// TwinCAT 3 PLC project TcoDrivesBeckhoff
// Title: TcoDrivesBeckhoff
// Company: Vortex.Library
// Author: TcOpenGroup
// ProjectVersion: 0.6.0.913
// ProgramVersion: 3.1.4024.12
// libraries:
//   Tc2_MC2, * (Beckhoff Automation GmbH)
//   Tc2_MC2_Drive, * (Beckhoff Automation GmbH)
//   Tc2_NCI, * (Beckhoff Automation GmbH)
//   Tc2_Standard, * (Beckhoff Automation GmbH)
//   Tc2_System, * (Beckhoff Automation GmbH)
//   Tc2_Utilities, * (Beckhoff Automation GmbH)
//   Tc3_Module, * (Beckhoff Automation GmbH)
//   TcoCore, 0.6.0.913 (Vortex.Library)
// project tree:
//   DUTs/ eAxisParameter.TcDUT (not stored), eAxisEncoderReferenceSystem.TcDUT (not stored), eDirection.TcDUT (not stored), eAxisStates.TcDUT (not stored), eEncoderReferenceMode.TcDUT (not stored), eHomingMode.TcDUT (not stored), ePowerOverride.TcDUT (not stored), eSetPositionMode.TcDUT (not stored), eJogMode.TcDUT (not stored), TcoAxisOpModes.TcDUT (not stored), TcoAxisRef.TcPOU (not stored), TcoAxisStatus.TcDUT (not stored), TcoAxisConfig.TcDUT (not stored)
//   DUTs/Interpolator/HW/ TcoGenericInterpolatorHw.TcDUT, TcoGenericInterpolatorHwInputs.TcDUT, TcoGenericInterpolatorHwOutputs.TcDUT
//   DUTs/Interpolator/ TcoGenericInterpolatorData.TcDUT
//   / PlcTask.TcTTO (not stored)
//   POUs/Conversions/ Tc2MC2_TO_Tco_AxisStates.TcPOU (not stored), LREAL_TO_Tco_AxisEncoderReferenceSystem.TcPOU (not stored), Tc2MC2_TO_Tco_SetPositionMode.TcPOU (not stored), Tc2MC2_TO_Tco_JogMode.TcPOU (not stored), Tco_TO_Tc2MC2_SetPositionMode.TcPOU (not stored), Tco_TO_Tc2MC2_Direction.TcPOU (not stored), Tc2MC2_TO_Tco_Direction.TcPOU (not stored), Tco_TO_Tc2MC2_HomingMode.TcPOU (not stored), Tco_TO_Tc2MC2_EncRefMode.TcPOU (not stored), Tc2MC2_TO_Tco_EncRefMode.TcPOU (not stored), Tc2MC2_TO_Tco_HomingMode.TcPOU (not stored), Tco_TO_Tc2MC2_AxisStates.TcPOU (not stored), Tco_TO_Tc2MC2_JogMode.TcPOU (not stored)
//   POUs/ MAIN.TcPOU (not stored)
//   POUs/Prototypes/CartesianCoordinateSystem/Intetrpolator/ TcoInterpolator.TcPOU, TcoInterpolatorConfig.TcDUT, TcoInterpolatorStatus.TcDUT, TcoInterpolatorControl.TcDUT
//   POUs/Prototypes/CartesianCoordinateSystem/MultiAxisSystem/ eTcoMultiAxisSystem.TcDUT (not stored), ITcoMultiAxis.TcIO (not stored), TcoMultiAxis.TcPOU (not stored), TcoMultiAxisConfig.TcDUT (not stored), TcoMultiAxisStatus.TcDUT (not stored), TcoMultiAxisMoveParam.TcDUT (not stored), TcoMultiAxisPositionsRootContainer.TcPOU (not stored)
//   POUs/Prototypes/CartesianCoordinateSystem/SingleAxisSystem/ ITcoSingleAxis.TcIO (not stored), TcoSingleAxisStatus.TcDUT (not stored), TcoSingleAxisConfig.TcDUT (not stored), TcoSingleAxis.TcPOU (not stored), TcoSingleAxisMoveParam.TcDUT (not stored), TcoSingleAxisPositionsRootContainer.TcPOU (not stored)
//   POUs/Prototypes/CartesianCoordinateSystem/ TcoAxisExchangeDataTask.TcPOU (not stored)
//   POUs/Prototypes/TcoDriveSimple/DriveState/ eTcoMovementState.TcDUT (not stored), TcoMovementState.TcPOU (not stored)
//   POUs/Prototypes/TcoDriveSimple/ ITcoDriveSimple.TcIO (not stored), Power.TcPOU (not stored), Jog.TcPOU (not stored), TcoDriveSimple.TcPOU (not stored)
//   POUs/Prototypes/TcoDriveSimple/MotionTasks/ HomeTask.TcPOU (not stored), MoveModuloTask.TcPOU (not stored), MoveRelativeTask.TcPOU (not stored), MoveAbsoluteTask.TcPOU (not stored), MoveVelocityTask.TcPOU (not stored), SetTorqueTask.TcPOU (not stored), StopTask.TcPOU (not stored), HaltTask.TcPOU (not stored)
//   POUs/Prototypes/TcoDriveSimple/AxisTasks/ ResetTask.TcPOU (not stored), SetPositionTask.TcPOU (not stored), SoEResetTask.TcPOU (not stored)

// ---- DUTs/Interpolator/HW/TcoGenericInterpolatorHw.TcDUT
TYPE TcoGenericInterpolatorHw :
STRUCT
	// In
	Inputs : TcoGenericInterpolatorHwInputs;

	// Out					
	Outputs : TcoGenericInterpolatorHwOutputs;
END_STRUCT
END_TYPE

// ---- DUTs/Interpolator/HW/TcoGenericInterpolatorHwInputs.TcDUT
TYPE TcoGenericInterpolatorHwInputs :
STRUCT
	iToPlc AT %I* : NCTOPLC_NCICHANNEL_REF;
END_STRUCT
END_TYPE

// ---- DUTs/Interpolator/HW/TcoGenericInterpolatorHwOutputs.TcDUT
TYPE TcoGenericInterpolatorHwOutputs :
STRUCT
	qFromPlc AT %Q* : PLCTONC_NCICHANNEL_REF;
END_STRUCT
END_TYPE

// ---- DUTs/Interpolator/TcoGenericInterpolatorData.TcDUT
{attribute addProperty Name "<#Data#>"}
{attribute wpf [Container(Layout.Stack)]}
TYPE TcoGenericInterpolatorData :
STRUCT

	{attribute addProperty Name "X - <#Actual Position#>"}
	posX : LREAL;
	{attribute addProperty Name "Y - <#Actual Position#>"}
	posY : LREAL;
	{attribute addProperty Name "Z - <#Actual Position#>"}
	posZ : LREAL;
	{attribute addProperty Name "<#Actual Interpolation Block No#>"}
	blockNo : UDINT;
	{attribute clr [ReadOnly()]}
	{attribute addProperty Name "<#Alarm Code#>"}
	AlarmCode : UDINT;
	
END_STRUCT
END_TYPE

// ---- POUs/Prototypes/CartesianCoordinateSystem/Intetrpolator/TcoInterpolatorConfig.TcDUT
TYPE TcoInterpolatorConfig :
STRUCT
   Axis1Disabled:BOOL;
   Axis2Disabled:BOOL;
   Axis3Disabled:BOOL;

   InfoTime : TIME := T#2S;
   ErrorTime : TIME := T#5S;
   
   Timeout:TIME :=T#15S;  
   FileName:STRING(254);  	
   Override : LREAL := 100.0;
   
  
END_STRUCT
END_TYPE

// ---- POUs/Prototypes/CartesianCoordinateSystem/Intetrpolator/TcoInterpolatorStatus.TcDUT
TYPE TcoInterpolatorStatus :
STRUCT
	ActionDescription : STRING(100);
	AlarmMessage : STRING(254);	
	Progress:int;
	Data: TcoGenericInterpolatorData;
END_STRUCT
END_TYPE

// ---- POUs/Prototypes/CartesianCoordinateSystem/Intetrpolator/TcoInterpolatorControl.TcDUT
TYPE TcoInterpolatorControl :
STRUCT
	{attribute addProperty Name "<#Velocity Override#>"}
	Override : LREAL := 100.0;
	{attribute addProperty Name "<#Interpolation File#>"}
	FileName : STRING;
END_STRUCT
END_TYPE

// ---- POUs/Prototypes/CartesianCoordinateSystem/Intetrpolator/TcoInterpolator.TcPOU
FUNCTION_BLOCK TcoInterpolator EXTENDS TcoCore.TcoComponent 
VAR_INPUT
	inEnableAxis1 : BOOL;
    inEnablePositiveAxis1 : BOOL;
    inEnableNegativeAxis1 : BOOL;
    inCalibrationCamAxis1 : BOOL;
	refAxis1 : REFERENCE TO TcoAxisRef;
	inEnableAxis2 : BOOL;
    inEnablePositiveAxis2 : BOOL;
    inEnableNegativeAxis2 : BOOL;
    inCalibrationCamAxis2 : BOOL;
	refAxis2 : REFERENCE TO TcoAxisRef;
	inEnableAxis3 : BOOL;
    inEnablePositiveAxis3 : BOOL;
    inEnableNegativeAxis3 : BOOL;
    inCalibrationCamAxis3 : BOOL;
	refAxis3 : REFERENCE TO TcoAxisRef;

END_VAR
VAR_IN_OUT
	IoData : TcoGenericInterpolatorHw;
END_VAR

VAR
	{attribute 'hide'}
    _axis1Ref : REFERENCE TO TcoAxisRef;
	{attribute addProperty Name "<#Axis 1#>"}
	_axis1 :   TcoDriveSimple(THIS^);
	{attribute 'hide'}
    _axis2Ref : REFERENCE TO TcoAxisRef;
	{attribute addProperty Name "<#Axis 2#>"}
	_axis2 :   TcoDriveSimple(THIS^);
	{attribute 'hide'}
    _axis3Ref : REFERENCE TO TcoAxisRef;
	{attribute addProperty Name "<#Axis 3#>"}
	_axis3 :   TcoDriveSimple(THIS^);

	
	interpBuildGroup		: Tc2_NCI.CfgBuild3DGroup;
	interpLoadGCode			: Tc2_NCI.ItpLoadProgEx;
	interpStartGCode		: Tc2_NCI.ItpStartStopEx;
	interpSingleBlock		: Tc2_NCI.ItpSingleBlock;
	interpClearGroup		: Tc2_NCI.CfgReconfigGroup;
	interpConfirmHsk		: Tc2_NCI.ItpConfirmHsk;
	interpReset				: Tc2_NCI.ItpResetEx2;
	
	
	{attribute addProperty Name "<#Status#>"}
    {attribute clr [ReadOnly()]}
    _status : TcoInterpolatorStatus;
	{attribute addProperty Name "<#Config#>"}
    _config : TcoInterpolatorConfig;
	{attribute addProperty Name "<#Control#>"}
    _control : TcoInterpolatorControl;
	
	
	
	{attribute addProperty Name "<#Start Interpolation#>"}
	_startInterpolation :   TcoCore.TcoTask (THIS^);
	
    {attribute addProperty Name "<#Block Mode#>"}
	{attribute addProperty StateOnDesc "<#On#>"}
	{attribute addProperty StateOffDesc "<#Off#>"}

	_blockMode :   TcoCore.TcoToggleTask(THIS^, FALSE);
	
	{attribute addProperty Name "<#Start Ground#>"}
	_startGroundPos :   TcoCore.TcoTask (THIS^);
	
	{attribute addProperty Name "<#Next step#>"}
	_nextStep :   TcoCore.TcoTask (THIS^);
	


	{attribute addProperty Name "<#Reset Drives Task#>"}
	_resetDrivesTask :   TcoCore.TcoTask (THIS^);
	{attribute addProperty Name "<#Soe Reset Drives Task#>"}
	_soeResetDrivesTask :   TcoCore.TcoTask (THIS^);

	{attribute addProperty Name "<#Restore Task#>"}
	_restoreTask :   TcoCore.TcoTask (THIS^);


	  {attribute 'hide'} 
	_infoTimer :  TON;
    {attribute 'hide'} 
	_errorTimer :  TON;
	_done: BOOL;
	_override: LREAL;
	
	{attribute clr [RenderIgnore()]}
	_fileOpened : BOOL;
    {attribute clr [RenderIgnore()]}
	_interpreterState : UDINT;
    {attribute clr [RenderIgnore()]}
	_hasError : BOOL;
	 {attribute 'hide'} 
	_progress: INT;
END_VAR






//*************RESTORE********************

_restoreTask.Enabled := TRUE;
IF _restoreTask.Execute() THEN
	Restore();
END_IF
//****************************************


IF NOT __ISVALIDREF(refAxis1)  AND NOT _config.Axis1Disabled THEN
    Messenger.Post('<#Invalid reference axis 1#>', TcoCore.eMessageCategory.ProgrammingError);
    RETURN;
ELSIF NOT _config.Axis1Disabled THEN
	_axis1Ref REF= refAxis1;


	_axis1(
		inEnable:=inEnableAxis1 , 
		inEnablePositive:=inEnablePositiveAxis1 , 
		inEnableNegative:=inEnableNegativeAxis1 , 
		inCalibrationCam:=inCalibrationCamAxis1, 
		inoAxisRef:= _axis1Ref);
END_IF


IF NOT __ISVALIDREF(refAxis2) AND NOT _config.Axis2Disabled THEN
    Messenger.Post('<#Invalid reference axis 2#>', TcoCore.eMessageCategory.ProgrammingError);
    RETURN;
ELSIF  NOT _config.Axis2Disabled THEN
	_axis2Ref REF= refAxis2;

	_axis2(
		inEnable:=inEnableAxis2 , 
		inEnablePositive:=inEnablePositiveAxis2 , 
		inEnableNegative:=inEnableNegativeAxis2 , 
		inCalibrationCam:=inCalibrationCamAxis2, 
		inoAxisRef:= _axis2Ref);
END_IF


IF NOT __ISVALIDREF(refAxis3) AND NOT _config.Axis3Disabled THEN
    Messenger.Post('<#Invalid reference axis 3#>', TcoCore.eMessageCategory.ProgrammingError);
    RETURN;
ELSIF NOT _config.Axis3Disabled THEN
	_axis3Ref REF= refAxis3;

	_axis3(
		inEnable:=inEnableAxis3 , 
		inEnablePositive:=inEnablePositiveAxis3 , 
		inEnableNegative:=inEnableNegativeAxis3 , 
		inCalibrationCam:=inCalibrationCamAxis3, 
		inoAxisRef:= _axis3Ref);
END_IF	

	




//*************Reset Drives********************

_resetDrivesTask.Enabled:= NOT _soeResetDrivesTask.Busy;
IF _resetDrivesTask.Execute() THEN
	

	IF  NOT _config.Axis1Disabled THEN 
		THIS^._axis1.Reset();
	END_IF;
	IF  NOT _config.Axis2Disabled THEN 
		THIS^._axis2.Reset();
	END_IF;
	IF  NOT _config.Axis3Disabled THEN 
		THIS^._axis3.Reset();
	END_IF;
	

	
	_hasError :=   (THIS^._axis1.ResetTask.Error AND NOT _config.Axis1Disabled)
				OR (THIS^._axis2.ResetTask.Error AND NOT _config.Axis2Disabled)
				OR (THIS^._axis3.ResetTask.Error AND NOT _config.Axis3Disabled) ;
	_done:=  (THIS^._axis1.ResetTask.Done XOR _config.Axis1Disabled)
		AND (THIS^._axis2.ResetTask.Done XOR _config.Axis2Disabled)
		AND (THIS^._axis3.ResetTask.Done XOR _config.Axis3Disabled);
			
		
	_resetDrivesTask.DoneWhen(_done);
	_resetDrivesTask.ThrowWhen(_hasError);	

END_IF;



_soeResetDrivesTask.Enabled:=  NOT _ResetDrivesTask.Busy;

//*************Soe Reset Drives********************
IF _soeResetDrivesTask.Execute() THEN
	
		IF  NOT _config.Axis1Disabled THEN 
			THIS^._axis1.SoEReset();
		END_IF;
		IF  NOT _config.Axis2Disabled THEN 
			THIS^._axis2.SoeReset();
		END_IF;
		IF  NOT _config.Axis3Disabled THEN 
			THIS^._axis3.SoEReset();
		END_IF;
		
				


		_hasError :=   (THIS^._axis1.SoEResetTask.Error AND NOT _config.Axis1Disabled)
					OR (THIS^._axis2.SoEResetTask.Error AND NOT _config.Axis2Disabled)
					OR (THIS^._axis3.SoEResetTask.Error AND NOT _config.Axis3Disabled)  ;
				
		_done:= (THIS^._axis1.SoEResetTask.Done XOR _config.Axis1Disabled)
			AND (THIS^._axis2.SoEResetTask.Done XOR _config.Axis2Disabled)
			AND (THIS^._axis3.SoEResetTask.Done XOR _config.Axis3Disabled);

	_soeResetDrivesTask.DoneWhen(_done);
	_soeResetDrivesTask.ThrowWhen(_errorTimer.Q OR _hasError);	
END_IF;

	
_startInterpolation.Enabled:=NOT _startGroundPos.Busy;	
IF _startInterpolation.Execute() THEN
	StartInterpolation(refProgress:=_progress, refTask:=_startInterpolation);
END_IF;	

_startGroundPos.Enabled:=NOT _startInterpolation.Busy;	
IF _startGroundPos.Execute() THEN
	GroundPosition(refProgress:=_progress,refTask:=_startGroundPos);
END_IF;	
	
//*************Block Mode********************
_blockMode.Enabled := THIS^.IsService;
_blockMode.Run();

IF _blockMode.IsOn THEN
		// activate single block mode
	THIS^.interpSingleBlock.nMode := E_ItpSingleBlockMode.ItpSingleBlockIntp;
	THIS^.interpSingleBlock.bTriggerNext := FALSE;
ELSE
		// deactivate single block mode
	THIS^.interpSingleBlock.nMode := E_ItpSingleBlockMode.ItpSingleBlockOff;
	THIS^.interpSingleBlock.bTriggerNext := FALSE;
END_IF;	


IF THIS^._blockMode.IsOn THEN 
	IF THIS^._nextStep.Execute() THEN
		THIS^.interpSingleBlock.bTriggerNext := TRUE;
		THIS^._nextStep.DoneWhen(TRUE);
	END_IF
ELSE
	THIS^._nextStep.Restore();
END_IF
ItpSetOverridePercent(fOverridePercent:= _control.Override , sPlcToNci:=THIS^.IoData.Outputs.qFromPlc);


THIS^.interpBuildGroup(
	bExecute:= , 
	nGroupId:= ItpGetGroupId(sNciToPlc:=THIS^.IoData.Inputs.iToPlc), 
	nXAxisId:= THIS^._axis1.AxisRef.NcToPlc.AxisId, 
	nYAxisId:= THIS^._axis2.AxisRef.NcToPlc.AxisId, 
	nZAxisId:= THIS^._axis3.AxisRef.NcToPlc.AxisId, 
	tTimeOut:= THIS^._config.Timeout, 
	bBusy=> , 
	bErr=> , 
	nErrId=> );

	
IF interpBuildGroup.bErr THEN
	Messenger.Error(CONCAT('<#Error executing Build Interpolation Group command. ErrorID:#> 0x',DWORD_TO_HEXSTR(UDINT_TO_DWORD(interpBuildGroup.nErrId),4,FALSE)));
END_IF

THIS^.interpLoadGCode(
	sNciToPlc:= THIS^.IoData.Inputs.iToPlc, 
	bExecute:= , 
	sPrg:= _control.FileName, 
	nLength:= INT_TO_UDINT(LEN(_control.FileName)), 
	tTimeOut:= Config.Timeout, 
	bBusy=> , 
	bErr=> , 
	nErrId=> );
	
IF interpLoadGCode.bErr THEN
	Messenger.Error(CONCAT('<#Error executing Load Program command. ErrorID:#> 0x',DWORD_TO_HEXSTR(UDINT_TO_DWORD(interpLoadGCode.nErrId),4,FALSE)));
END_IF
	
THIS^.interpStartGCode(
	bStart:= , 
	bStop:= , 
	tTimeOut:= Config.Timeout, 
	sNciToPlc:= THIS^.IoData.Inputs.iToPlc, 
	bBusy=> , 
	bErr=> , 
	nErrId=> );
	
IF interpStartGCode.bErr THEN
	Messenger.Error(CONCAT('<#Error executing Start Program command. ErrorID:#> 0x',DWORD_TO_HEXSTR(UDINT_TO_DWORD(interpStartGCode.nErrId),4,FALSE)));
END_IF

THIS^.interpSingleBlock(
	bExecuteModeChange:= , 
	nMode:= , 
	bTriggerNext:= , 
	tTimeOut:= Config.Timeout, 
	sNciToPlc:= THIS^.IoData.Inputs.iToPlc, 
	bBusy=> , 
	bErr=> , 
	nErrId=> );

THIS^.interpClearGroup(
	bExecute:= , 
	nGroupId:= ItpGetGroupId(sNciToPlc:=THIS^.IoData.Inputs.iToPlc), 
	tTimeOut:= Config.Timeout, 
	bBusy=> , 
	bErr=> , 
	nErrId=> );
	
IF interpClearGroup.bErr THEN
	Messenger.Error(CONCAT('<#Error executing Clear Group command. ErrorID:#> 0x',DWORD_TO_HEXSTR(UDINT_TO_DWORD(interpClearGroup.nErrId),4,FALSE)));
END_IF

THIS^.interpConfirmHsk(
	bExecute:= , 
	sNciToPlc:= THIS^.IoData.Inputs.iToPlc, 
	sPlcToNci:= THIS^.IoData.Outputs.qFromPlc, 
	bBusy=> , 
	bErr=> , 
	nErrId=> );

IF interpConfirmHsk.bErr THEN
	Messenger.Error(CONCAT('<#Error executing Confirm Handshake command. ErrorID:#> 0x',DWORD_TO_HEXSTR(UDINT_TO_DWORD(interpConfirmHsk.nErrId),4,FALSE)));
END_IF

THIS^.interpReset(
	bExecute:= , 
	tTimeOut:= Config.Timeout, 
	sNciToPlc:= THIS^.IoData.Inputs.iToPlc, 
	bBusy=> , 
	bErr=> , 
	nErrId=> );
	
_status.Progress:=_progress;
_status.Data.posX:=_axis1.AxisStatus.ActPos;
_status.Data.posY:=_axis2.AxisStatus.ActPos;
_status.Data.posZ:=_axis3.AxisStatus.ActPos;
_status.Data.blockNo := ItpGetBlockNumber(sNciToPlc := THIS^.IoData.Inputs.iToPlc);
_status.Data.AlarmCode := ItpGetError(sNciToPlc := THIS^.IoData.Inputs.iToPlc);
	
IF interpReset.bErr THEN
	Messenger.Error(CONCAT('<#Error executing Reset command#>: ',DWORD_TO_HEXSTR(UDINT_TO_DWORD(interpReset.nErrId),4,TRUE)));
END_IF


THIS^._interpreterState := ItpGetStateInterpreter(sNciToPlc:=THIS^.IoData.Inputs.iToPlc);

THIS^._hasError := interpBuildGroup.bErr OR interpLoadGCode.bErr OR interpStartGCode.bErr;

Messenger.OnCondition(Status.Data.AlarmCode <> 0).Error(  THIS^.GetErrorDescription());

PROPERTY Axis_1 : REFERENCE TO TcoDriveSimple
GET
Axis_1 REF=_axis1;
END_GET
END_PROPERTY

PROPERTY Axis_2 : REFERENCE TO TcoDriveSimple
GET
Axis_2 REF=_axis2;
END_GET
END_PROPERTY

PROPERTY Axis_3 : REFERENCE TO TcoDriveSimple
GET
Axis_3 REF=_axis3;
END_GET
END_PROPERTY

METHOD CallTimers
VAR_INPUT
	inValue : BOOL;
END_VAR
IF  __ISVALIDREF(Config) THEN  
_infoTimer(IN := inValue, PT := THIS^.Config.InfoTime);
_errorTimer(IN := inValue, PT := THIS^.Config.ErrorTime);
END_IF;
END_METHOD

(*~
	<docu>
		<summary>
			Gets the configuration of the interpolator. 					
		</summary>			
	</docu>	
~*)
PROPERTY Config : REFERENCE TO TcoInterpolatorConfig
GET
Config REF= _config;
END_GET
END_PROPERTY

METHOD GetErrorDescription : STRING(254)
VAR_INPUT
END_VAR
VAR
	status:STRING(254);
END_VAR
_status.AlarmMessage := '';


CASE _status.Data.AlarmCode OF
	0: status := 'No Error';
	16#4000 .. 16#40FF: status := CONCAT(DWORD_TO_HEXSTR((_status.Data.AlarmCode),4,FALSE),' - <#General Error#> - <#see detailed description in Component View#>');
	16#4100 .. 16#41FF: status := CONCAT(DWORD_TO_HEXSTR((_status.Data.AlarmCode),4,FALSE),' - <#Channel Error#> - <#see detailed description in Component View#>');
	16#4200 .. 16#42FF: status := CONCAT(DWORD_TO_HEXSTR((_status.Data.AlarmCode),4,FALSE),' - <#Group Error#> - <#see detailed description in Component View#>');
	16#4300 .. 16#43FF: status := CONCAT(DWORD_TO_HEXSTR((_status.Data.AlarmCode),4,FALSE),' - <#Axis Error#> - <#see detailed description in Component View#>');
	16#4400 .. 16#44FF: status := CONCAT(DWORD_TO_HEXSTR((_status.Data.AlarmCode),4,FALSE),' - <#Encoder Error#> - <#see detailed description in Component View#>');
	16#4500 .. 16#45FF: status := CONCAT(DWORD_TO_HEXSTR((_status.Data.AlarmCode),4,FALSE),' - <#Controller Error#> - <#see detailed description in Component View#>');
	16#4600 .. 16#46FF: status := CONCAT(DWORD_TO_HEXSTR((_status.Data.AlarmCode),4,FALSE),' - <#Drive Error#> - <#see detailed description in Component View#>');
	16#4A00 .. 16#4AFF: status := CONCAT(DWORD_TO_HEXSTR((_status.Data.AlarmCode),4,FALSE),' - <#Table Error#> - <#see detailed description in Component View#>');
	16#4B00 .. 16#4BFF: status := CONCAT(DWORD_TO_HEXSTR((_status.Data.AlarmCode),4,FALSE),' - <#NC PLC Error#> - <#see detailed description in Component View#>');
	16#4C00 .. 16#4CFF: status := CONCAT(DWORD_TO_HEXSTR((_status.Data.AlarmCode),4,FALSE),' - <#Kinematic Transformation Error#> - <#see detailed description in Component View#>');
	16#8100 .. 16#811F: status := CONCAT(DWORD_TO_HEXSTR((_status.Data.AlarmCode),4,FALSE),' - <#Bode Plot Error#> - <#see detailed description in Component View#>');
	16#8120 .. 16#8FFF: status := CONCAT(DWORD_TO_HEXSTR((_status.Data.AlarmCode),4,FALSE),' - <#Furhter Error#> - <#see detailed description in Component View#>');
	
ELSE
	status := 'Unknown Error';
END_CASE
_status.AlarmMessage :=status;
GetErrorDescription := status;
END_METHOD

METHOD PUBLIC Ground : TcoCore.ITcoTaskStatus
Ground:=THIS^._startGroundPos.Invoke();
END_METHOD

(*

			DESCRIBE FUNCTION OF THIS METHOD

*)
METHOD PRIVATE GroundPosition
VAR_INPUT
    refProgress : REFERENCE TO INT;
    refTask : REFERENCE TO TcoCore.TcoTask;
END_VAR
VAR_INST
    _progress : REFERENCE TO INT;
    _task : REFERENCE TO TcoCore.TcoTask;
END_VAR
_progress REF= refProgress;
_task REF= refTask;


IF _progress = 0 THEN
//--------------------------------------------------------------  
	interpStartGCode.bStop := TRUE;
	_status.ActionDescription:='Waiting to  Tc2_NCI.NCI_INTERPRETER_IDLE';
	IF _interpreterState = Tc2_NCI.NCI_INTERPRETER_IDLE THEN	
		interpStartGCode.bStop := FALSE;		
		_progress := 10;
	ELSE
		Messenger.Info('<#Interpreter not in IDLE state.#>');
	END_IF
//--------------------------------------------------------------  
END_IF

IF _progress = 10 THEN
//--------------------------------------------------------------   
	interpReset.bExecute := TRUE;
	_status.ActionDescription:='Waiting to interpReset.bBusy';

	IF (interpReset.bBusy) THEN
		_progress := _progress + 1;
	END_IF
//--------------------------------------------------------------	
END_IF

IF _progress = 11 THEN
//--------------------------------------------------------------
	_status.ActionDescription:='Waiting to NOT interpReset.bBusy';   
	IF NOT interpReset.bBusy THEN
		interpReset.bExecute := FALSE;
		_progress := _progress + 1;
	END_IF
//--------------------------------------------------------------	
END_IF

IF _progress = 12 THEN
//--------------------------------------------------------------   
	interpClearGroup.bExecute := TRUE;
	_status.ActionDescription:='Waiting to interpClearGroup.bBusy';
	IF (interpClearGroup.bBusy) THEN
		_progress := _progress + 1;
	END_IF
//--------------------------------------------------------------	
END_IF

IF _progress = 13 THEN
//--------------------------------------------------------------   
	_status.ActionDescription:='Waiting to NOT interpClearGroup.bBusy';
	IF NOT interpClearGroup.bBusy AND NOT interpClearGroup.bErr THEN	
		interpClearGroup.bExecute := FALSE;		
		_progress := _progress + 1;
	END_IF
//--------------------------------------------------------------	
END_IF

IF _progress = 14 THEN
//--------------------------------------------------------------   
_task.DoneWhen(TRUE);
//--------------------------------------------------------------	
END_IF

_task.ThrowWhen(_task.ElapsedTime>_config.ErrorTime);
Messenger.OnCondition(_infoTimer.Q AND _status.ActionDescription<>'').Info(concat(TO_STRING(_progress), _status.ActionDescription));
END_METHOD

METHOD Handshake
VAR_IN_OUT
	iHandshakeAck : BOOL;
	qHandshake : BOOL;
END_VAR
// all m-functions are directly confiremd. In a real application we have of course to consider the m-function numbers to turn on/off certain functions in the machine.
IF ItpIsHskMFunc(THIS^.IoData.Inputs.iToPlc) AND NOT interpConfirmHsk.bBusy THEN
	qHandshake := TRUE;
	IF iHandshakeAck THEN
		interpConfirmHsk.bExecute	:= TRUE;
	END_IF
ELSE	
	qHandshake := FALSE;
	interpConfirmHsk.bExecute	:= FALSE;
END_IF
END_METHOD

METHOD PUBLIC Interpolate : TcoCore.ITcoTaskStatus
_control.FileName:=_config.FileName;
_control.Override:=_config.Override;


Interpolate:=THIS^._startInterpolation.Invoke();
END_METHOD

(*

			DESCRIBE FUNCTION OF THIS METHOD

*)
METHOD InterpolateWithHandshake : TcoCore.ITcoTaskStatus
VAR_INPUT
	inFileName : STRING;
	inOverride : LREAL;
END_VAR
VAR_IN_OUT
	inoIHandshakeAck : BOOL;
	inoQHandshake : BOOL;
END_VAR
_control.FileName:=inFileName;
_control.Override:=inOverride;

InterpolateWithHandshake:=THIS^._startInterpolation.Invoke();

// all m-functions are directly confiremd. In a real application we have of course to consider the m-function numbers to turn on/off certain functions in the machine.
Handshake(inoIHandshakeAck,inoQHandshake);	

// Hlasenie o stave priebehu volania metody
//THIS^._progressMessage.Post(Message:= CONCAT('@en-US@Executing action ~', INT_TO_STRING(THIS^._progress)), Category:= enumMessageCategory.Info);
END_METHOD

(*

			DESCRIBE FUNCTION OF THIS METHOD

*)
METHOD InterpolateWithHandshakeAndOutput : TcoCore.ITcoTaskStatus
VAR_INPUT
	inFileName : STRING;
	inOverride : LREAL;
END_VAR
VAR_IN_OUT
	inoIHandshakeAck : BOOL;
	inoQHandshake : BOOL;
	inoProgrammedOutput : BOOL;
END_VAR
_control.FileName:=inFileName;
_control.Override:=inOverride;

InterpolateWithHandshakeAndOutput:=THIS^._startInterpolation.Invoke();

// handling of m-functions is done outside statemachine
// M10 is signal for start and M11 is signal for stop
SetOutputWithMFunction(10,inoProgrammedOutput);
ResetOutputWithMFunction(11,inoProgrammedOutput);

// all m-functions are directly confiremd. In a real application we have of course to consider the m-function numbers to turn on/off certain functions in the machine.
Handshake(inoIHandshakeAck,inoQHandshake);	

// Hlasenie o stave priebehu volania metody
//THIS^._progressMessage.Post(Message:= CONCAT('@en-US@Executing action ~', INT_TO_STRING(THIS^._progress)), Category:= enumMessageCategory.Info);
END_METHOD

METHOD PUBLIC InterpolateWithParam : TcoCore.ITcoTaskStatus
VAR_INPUT
	inFileName : STRING;
	inOverride : LREAL;
END_VAR
_control.FileName:=inFileName;
_control.Override:=inOverride;

InterpolateWithParam:=THIS^._startInterpolation.Invoke();
END_METHOD

PROPERTY IsRunning : BOOL
GET
IsRunning := _interpreterState = Tc2_NCI.NCI_INTERPRETER_RUNNING;
END_GET
END_PROPERTY

METHOD ResetDrives : TcoCore.ITcoTaskStatus
ResetDrives:=THIS^._resetDrivesTask.Invoke();
END_METHOD

PROPERTY PUBLIC ResetDrivesTask : REFERENCE TO TcoCore.TcoTask
GET
ResetDrivesTask REF=_resetDrivesTask;
END_GET
END_PROPERTY

METHOD ResetOutputWithMFunction
VAR_INPUT
	MfunctionNo : INT;
END_VAR
VAR_IN_OUT
	programmedOutput : BOOL;
END_VAR
IF ItpIsFastMFunc(MfunctionNo,THIS^.IoData.Inputs.iToPlc) 
	OR NOT (_interpreterState = Tc2_NCI.NCI_INTERPRETER_RUNNING) THEN
	programmedOutput := FALSE;
END_IF;
END_METHOD

(*~
	<docu>
		<summary>
			Restores this instance to the Ready state. Can be called explicitly or from within one of the restore mechanisms.	
		</summary>			
	</docu>	
~*)
METHOD  Restore : ITcoRestorable
_axis1.Restore();
_axis2.Restore();
_axis3.Restore();
_restoreTask.Restore();

_progress:=0;
_soeResetDrivesTask.Restore();
_resetDrivesTask.Restore();
_startGroundPos.Restore();
_startInterpolation.Restore();
_nextStep.Restore();
CallTimers(FALSE);


// disable execute
interpBuildGroup.bExecute := FALSE;
interpClearGroup.bExecute := FALSE;
interpLoadGCode.bExecute := FALSE;
interpStartGCode.bStart := FALSE;
interpStartGCode.bStop := TRUE;
interpSingleBlock.bExecuteModeChange := FALSE;
interpSingleBlock.bTriggerNext := FALSE;
interpConfirmHsk.bExecute := FALSE;
interpReset.bExecute := FALSE;
interpSingleBlock.nMode := E_ItpSingleBlockMode.ItpSingleBlockOff;
Messenger.UnPin();
END_METHOD

METHOD PROTECTED ServiceMode
THIS^._axis1.Service();
THIS^._axis2.Service();
THIS^._axis3.Service();
END_METHOD

METHOD SetOutputWithMFunction
VAR_INPUT
	MfunctionNo : INT;
END_VAR
VAR_IN_OUT
	programmedOutput : BOOL;
END_VAR
IF ItpIsFastMFunc(MfunctionNo,THIS^.IoData.Inputs.iToPlc) THEN
	programmedOutput := TRUE;
END_IF;
END_METHOD

METHOD SoeReset : TcoCore.ITcoTaskStatus
SoeReset:=THIS^._soeResetDrivesTask.Invoke();
END_METHOD

PROPERTY PUBLIC SoeResetDrivesTask : REFERENCE TO TcoCore.TcoTask
GET
SoeResetDrivesTask REF=_soeResetDrivesTask;
END_GET
END_PROPERTY

(*

			DESCRIBE FUNCTION OF THIS METHOD

*)
METHOD PRIVATE StartInterpolation 
VAR_INPUT
	refProgress:REFERENCE TO INT;
	refTask:REFERENCE TO TcoCore.TcoTask;
END_VAR
VAR_INST
	_progress:REFERENCE TO INT;
	_task:REFERENCE TO TcoCore.TcoTask;
END_VAR
_progress REF= refProgress;
_task REF= refTask;

IF _progress = 0 THEN
    //--------------------------------------------------------------  
    // Inicializacia
    interpBuildGroup.bExecute := FALSE;
    interpLoadGCode.bExecute := FALSE;
    interpStartGCode.bStart := FALSE;
    interpStartGCode.bStop := FALSE;
    interpClearGroup.bExecute := FALSE;
    interpReset.bExecute := FALSE;
    interpSingleBlock.bExecuteModeChange := FALSE;

    IF LEN(_control.FileName) <= 0 THEN
        Messenger.Error('<#Invalid file name of interpolation file.#>');
    END_IF

    IF (NOT interpReset.bBusy AND LEN(_control.FileName) > 0) THEN
        _progress := 100;
    END_IF
    //--------------------------------------------------------------  
END_IF

IF _progress = 100 THEN
    //--------------------------------------------------------------   

    _progress := _progress + 1;

    //--------------------------------------------------------------	
END_IF

IF _progress = 101 THEN
    //--------------------------------------------------------------   
    interpReset.bExecute := TRUE;
    _status.ActionDescription := 'Waiting to interpReset.bBusy';

    IF interpReset.bBusy THEN
        _progress := _progress + 1;
    END_IF
    //--------------------------------------------------------------	
END_IF

IF _progress = 102 THEN
    //--------------------------------------------------------------   
    _status.ActionDescription := 'Waiting to NOT interpReset.bBusy';

    IF NOT interpReset.bBusy THEN
        interpReset.bExecute := FALSE;
        _progress := _progress + 1;
    END_IF

    //--------------------------------------------------------------	
END_IF

IF _progress = 103 THEN
    //--------------------------------------------------------------   
    interpBuildGroup.bExecute := TRUE;
    _status.ActionDescription := 'Waiting to interpBuildGroup.bBusy';

    IF interpBuildGroup.bBusy THEN
        _progress := _progress + 1;
    END_IF
    //--------------------------------------------------------------	
END_IF

IF _progress = 104 THEN
    //--------------------------------------------------------------   
    _status.ActionDescription := 'Waiting to NOT interpBuildGroup.bBusy';

    IF NOT interpBuildGroup.bBusy THEN
        interpBuildGroup.bExecute := FALSE;
        _progress := _progress + 1;
    END_IF

    //--------------------------------------------------------------	
END_IF

IF _progress = 105 THEN
    //--------------------------------------------------------------   
    interpLoadGCode.bExecute := TRUE;
    _status.ActionDescription := 'Waiting to interpLoadGCode.bBusy';

    IF interpLoadGCode.bBusy THEN
        _progress := _progress + 1;
    END_IF
    //--------------------------------------------------------------	
END_IF

IF _progress = 106 THEN
    //--------------------------------------------------------------   
    _status.ActionDescription := 'Waiting to NOT interpLoadGCode.bBusy and NOT interpLoadGCode.bErr ';

    IF NOT interpLoadGCode.bBusy AND NOT interpLoadGCode.bErr THEN
        interpLoadGCode.bExecute := FALSE;
        _progress := _progress + 1;
    END_IF

    //--------------------------------------------------------------	
END_IF

IF _progress = 107 THEN
    //--------------------------------------------------------------   
    _status.ActionDescription := 'Waiting to Tc2_NCI.NCI_INTERPRETER_READY';

    IF _interpreterState = Tc2_NCI.NCI_INTERPRETER_READY THEN
        _progress := _progress + 1;
    END_IF

    //--------------------------------------------------------------	
END_IF

IF _progress = 108 THEN
    //--------------------------------------------------------------   
    interpStartGCode.bStart := TRUE;
    interpStartGCode.bStop := FALSE;
    interpSingleBlock.bExecuteModeChange := TRUE;

    _status.ActionDescription := 'Waiting to interpStartGCode.bBusyY';

    IF interpStartGCode.bBusy THEN
        _progress := _progress + 1;
    END_IF
    //--------------------------------------------------------------	
END_IF

IF _progress = 109 THEN
    //--------------------------------------------------------------   
    _status.ActionDescription := 'Waiting to NOT interpStartGCode.bBusy AND NOT interpStartGCode.bErr ';

    IF NOT interpStartGCode.bBusy AND NOT interpStartGCode.bErr THEN
        interpStartGCode.bStart := FALSE;
        _progress := _progress + 1;
    END_IF

    //--------------------------------------------------------------	
END_IF

IF _progress = 110 THEN
    //--------------------------------------------------------------  
    _status.ActionDescription := 'Waiting to NOT Tc2_NCI.NCI_INTERPRETER_READY ';

    IF _interpreterState <> Tc2_NCI.NCI_INTERPRETER_READY THEN
        _progress := _progress + 1;
    END_IF

    //--------------------------------------------------------------	
END_IF

IF _progress = 111 THEN
    //-------------------------------------------------------------- 
    _status.ActionDescription := 'Waiting to Tc2_NCI.NCI_INTERPRETER_READY ';

    IF _interpreterState = Tc2_NCI.NCI_INTERPRETER_READY THEN
        _progress := _progress + 1;
    ELSIF _interpreterState = Tc2_NCI.NCI_INTERPRETER_ABORTED THEN
        Messenger.Error('<#Interpolácia prerušená.#>');
    END_IF

    //--------------------------------------------------------------	
END_IF

IF _progress = 112 THEN
    //--------------------------------------------------------------   
    interpClearGroup.bExecute := TRUE;
    _status.ActionDescription := 'Waiting to interpClearGroup.bBusy';

    IF interpClearGroup.bBusy THEN
        _progress := _progress + 1;
    END_IF
    //--------------------------------------------------------------	
END_IF

IF _progress = 113 THEN
    //--------------------------------------------------------------   
    _task.DoneWhen(TRUE);

    //--------------------------------------------------------------	
END_IF

_task.ThrowWhen(_task.ElapsedTime > _config.ErrorTime);
Messenger.OnCondition(_infoTimer.Q AND _status.ActionDescription <> '').Info(concat(TO_STRING(_progress), _status.ActionDescription));

// handling of m-functions is done outside statemachine
// M10 is signal for start and M11 is signal for stop
//IF ItpIsFastMFunc(10,THIS^.IoData.Inputs.iToPlc) THEN
//	programmedOutput := TRUE;
//END_IF

//IF ItpIsFastMFunc(11,THIS^.IoData.Inputs.iToPlc) THEN
//	programmedOutput := FALSE;
//END_IF

//// all m-functions are directly confiremd. In a real application we have of course to consider the m-function numbers to turn on/off certain functions in the machine.
//IF ItpIsHskMFunc(THIS^.IoData.Inputs.iToPlc) AND NOT interpConfirmHsk.bBusy THEN
//	interpConfirmHsk.bExecute	:= TRUE;
//ELSE	
//	interpConfirmHsk.bExecute	:= FALSE;
//END_IF	

// Hlasenie o stave priebehu volania metody
//THIS^._progressMessage.Post(Message:= CONCAT('@en-US@Executing action ~', INT_TO_STRING(THIS^._progress)), Category:= enumMessageCategory.Info);
END_METHOD

(*~
	<docu>
		<summary>
			Gets the status of the Interpolator 					
		</summary>			
	</docu>	
~*)
PROPERTY Status : REFERENCE TO TcoInterpolatorStatus
GET
Status REF= _status;
END_GET
END_PROPERTY

END_FUNCTION_BLOCK
